# EPICS substitutions: epics/db/EL5021.substitutions
file "./db/ecSlave.template"
{
  pattern {}
          {}
}

#file "./db/EL5021.template"
#{
#  pattern {CH_ID, LINR,    ESLO,   EOFF,   EGU,        PREC, LOW, LOLO, HIGH, HIHI, HYST, LLSV,       LSV,        HSV,        HHSV      }
#          {1,     "SLOPE", 0.1,    0,      "DegC",     0,    0,   0,    0,    0,    0,    "NO_ALARM", "NO_ALARM", "NO_ALARM", "NO_ALARM"}
#}
